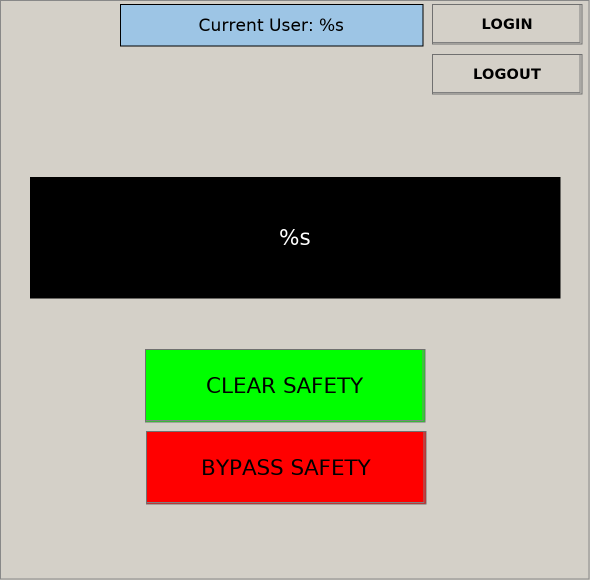
VISUALIZATION safetyResetScreen  // 590x580
    Rectangle (30,177 530x121), "%s", text variable: MAIN.sSafetyResetMsg
    Button (145,349 280x73), "CLEAR SAFETY"
        toggle MAIN.bSafetyResetBtn
    Button (146,431 280x73), "BYPASS SAFETY"
        toggle GVL_machine.bSafetyBypass
        OnMouseDown: execute {
            IF NOT GVL_devices.fbEstop.bEstopSigOk THEN
            	main.bBypassResetEstop := TRUE;
            END_IF
        }
    Button (432,4 150x40), "LOGIN"
        OnMouseDown: VisuUserMgmt Type=Login
    Button (432,54 150x40), "LOGOUT"
        OnMouseDown: VisuUserMgmt Type=Logout
    Textfield (120,4 303x42), "Current User: %s", text variable: VisuElems.CurrentUserName
END_VISUALIZATION

(* stored: Version 1.1.0.1, ProductVersion 3.1.4024.13
   Visu safetyResetScreen: Id {95c16017-7a82-48dc-8818-38289da7917b} *)
